TYPE mbar : REAL; END_TYPE

(* stored: Version 1.1.0.1, ProductVersion 3.1.4024.4
   DUT mbar: Id {389c2bb2-dc0e-46af-a085-473e48de876f} *)
